// TIA Portal V17 export
// export: Created 2025-03-07T09:17:56.294685Z, ExportSetting WithDefaults, DisplayName Totally Integrated Automation Portal, DisplayVersion V17 Update 8, DisplayName TIA Portal Openness, DisplayVersion V17 Update 8, DisplayName TIA Portal Version Control Interface, DisplayVersion V17, DisplayName SINAMICS Startdrive Advanced, DisplayVersion V17 SP2, DisplayName SINAMICS Startdrive G110M, G120, G120C, G120D, G120P, G115D, DisplayVersion V17 SP2, DisplayName SINAMICS Startdrive G130, G150, S120, S150, SINAMICS MV, S210, DisplayVersion V17 SP2, DisplayName STEP 7 Professional, DisplayVersion V17 Update 8, DisplayName SINUMERIK ONE STEP 7 Toolbox, DisplayVersion V17 Update 12, DisplayName SINUMERIK 840D sl STEP 7 Toolbox, DisplayVersion V17 Update 12, DisplayName STEP 7 Safety, DisplayVersion V17 Update 6, DisplayName WinCC Advanced, DisplayVersion V17 Update 8
FUNCTION "FC1100_MAIN_SEQUENCES" : Void   // FC1100, LAD
{ S7_Optimized_Access := 'FALSE' }
AUTHOR : ETXETAR
VERSION : 1.0
// stored: AutoNumber false, IsIECCheckEnabled false, SetENOAutomatically false, UDAEnableTagReadback false
   VAR_TEMP
      STEP_NUMBER : Int;
   END_VAR
BEGIN

REGION Network 1: CALL FC1103 MACHINING TWIN TWIN+
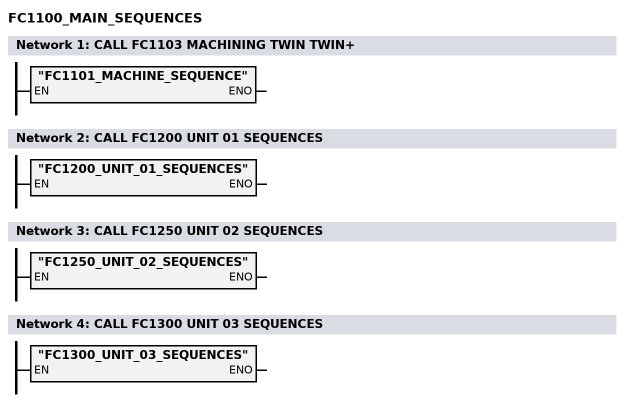
   RUNG wire#powerrail
      "FC1101_MACHINE_SEQUENCE"()
   END_RUNG
   // the same network as SCL:
   "FC1101_MACHINE_SEQUENCE"();
END_REGION

REGION Network 2: CALL FC1200 UNIT 01 SEQUENCES
   RUNG wire#powerrail
      "FC1200_UNIT_01_SEQUENCES"()
   END_RUNG
   // the same network as SCL:
   "FC1200_UNIT_01_SEQUENCES"();
END_REGION

REGION Network 3: CALL FC1250 UNIT 02 SEQUENCES
   RUNG wire#powerrail
      "FC1250_UNIT_02_SEQUENCES"()
   END_RUNG
   // the same network as SCL:
   "FC1250_UNIT_02_SEQUENCES"();
END_REGION

REGION Network 4: CALL FC1300 UNIT 03 SEQUENCES
   RUNG wire#powerrail
      "FC1300_UNIT_03_SEQUENCES"()
   END_RUNG
   // the same network as SCL:
   "FC1300_UNIT_03_SEQUENCES"();
END_REGION
END_FUNCTION
